// TIA Portal V19 export
FUNCTION_BLOCK "LAF_PowerOnOff"   // FB28, LAD
TITLE = LAF_ControlOnOff
AUTHOR : Siemens Digital Industries
FAMILY : LAF
VERSION : 1.0
// Control and managment of the power on/off of the system
// stored: Access Published, IsIECCheckEnabled true, MemoryReserve 100, SetENOAutomatically true
   VAR_INPUT
      on : Bool;   // Command to turn on
      off : Bool;   // Command to turn off
   END_VAR
   VAR_OUTPUT
      powerStatus { ExternalWritable := 'False'} : Int;   // 0 - Off, 1 - Paused, 2 - On
   END_VAR
   VAR_IN_OUT
      enablePower { ExternalWritable := 'False'} : Bool;   // Current power status
   END_VAR
   VAR
      statMemOn { ExternalWritable := 'False'} : Bool;   // Saved power status of last cycle
   END_VAR
   VAR CONSTANT
      POWER_STATUS_OFF : Int := 0;   // ID for Power off
      POWER_STATUS_PAUSED : Int := 1;   // ID for Power Paused
      POWER_STATUS_ON : Int := 2;   // ID for Power on
   END_VAR
   VAR_TEMP   // added for the SCL form of the ladder/FBD networks
      _w1 : Bool;
   END_VAR
BEGIN

REGION Network 1: BLOCK INFO HEADER
   // SIEMENS AG / (c)Copyright 2024
   // ------------------------------------------------------------------------------
   // Title:            LAF_ControlOnOff
   // Comment/Function: Control and managment of the power on/off of the system
   // Library/Family:   Library of Automation Framework
   // Author:                Siemens Digital Industry
   // Tested with:       S7-PLCSIM Advanced 6.0
   // Engineering:      TIA Portal V19
   // Restrictions:       ---
   // Requirements:   ---
   // ------------------------------------------------------------------------------
   // Change log table:
   // Version  | Date       | Expert in charge       | Changes applied
   // ---------|------------|------------------------|------------------------------
   // 01.01.00 | 21.06.2024 | SIMATIC Systems Support
   //                         First released version
   // 01.02.00 | 23.09.2024 | SIMATIC Systems Support
   //                         Block information properties updated
   //                         Changed input enablePower to an inOut and adjusted program
END_REGION

REGION Network 2: DESCRIPTION
   // This block controls the powered on /off status of a system. 
   // 1. Power On: The system will have the status power on in case it recieves an _on_ (any customized condition) input. 
   // 2. Power Off: The system will have the status power off in case it recieves an _off_ (any customized condition) input.
END_REGION

REGION Network 3: Evaluate commands
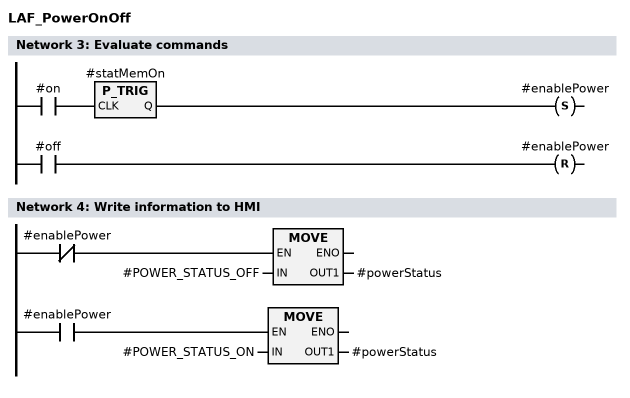
   RUNG wire#powerrail
      Contact( #on )
      P_Trig( #statMemOn )
      S_Coil( #enablePower )
   END_RUNG
   RUNG wire#powerrail
      Contact( #off )
      R_Coil( #enablePower )
   END_RUNG
   // the same network as SCL:
   #_w1 := #on AND NOT #statMemOn;   // rising edge
   #statMemOn := #on;
   IF #_w1 THEN #enablePower := TRUE; END_IF;
   IF #off THEN #enablePower := FALSE; END_IF;
END_REGION

REGION Network 4: Write information to HMI
   RUNG wire#powerrail
      I_Contact( #enablePower )
      Move(in := #POWER_STATUS_OFF, out1 => #powerStatus)
   END_RUNG
   RUNG wire#powerrail
      Contact( #enablePower )
      Move(in := #POWER_STATUS_ON, out1 => #powerStatus)
   END_RUNG
   // the same network as SCL:
   IF NOT #enablePower THEN #powerStatus := #POWER_STATUS_OFF; END_IF;
   IF #enablePower THEN #powerStatus := #POWER_STATUS_ON; END_IF;
END_REGION
END_FUNCTION_BLOCK
